// LS Electric XG5000 project: 과년66_1_1
// PLC NewPLC
// module base 0 slot 0: 입출력 모듈:XBC-DR20S (DC 24V 입력 12점, 릴레이 출력 8점)

PROGRAM NewProgram (task: 스캔 프로그램)

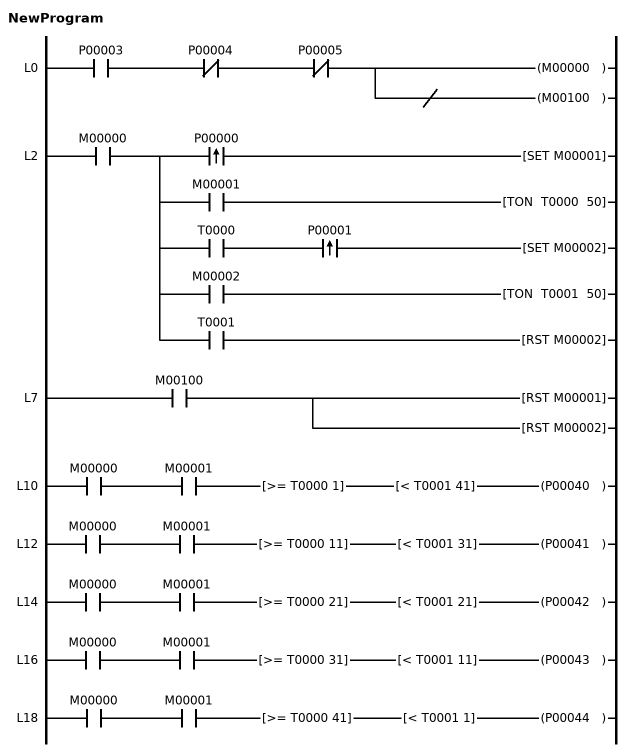
; L0
LOAD      P00003
AND NOT   P00004
AND NOT   P00005
OUT       M00000
NOT
OUT       M00100
; L2
LOAD      M00000
MPUSH
ANDP      P00000
SET       M00001
MLOAD
AND       M00001
TON       T0000 50
MLOAD
AND       T0000
ANDP      P00001
SET       M00002
MLOAD
AND       M00002
TON       T0001 50
MPOP
AND       T0001
RST       M00002
; L7
LOAD      M00100
RST       M00001
RST       M00002
; L10
LOAD      M00000
AND       M00001
AND>=     T0000 1
AND<      T0001 41
OUT       P00040
; L12
LOAD      M00000
AND       M00001
AND>=     T0000 11
AND<      T0001 31
OUT       P00041
; L14
LOAD      M00000
AND       M00001
AND>=     T0000 21
AND<      T0001 21
OUT       P00042
; L16
LOAD      M00000
AND       M00001
AND>=     T0000 31
AND<      T0001 11
OUT       P00043
; L18
LOAD      M00000
AND       M00001
AND>=     T0000 41
AND<      T0001 1
OUT       P00044